PROGRAM MAIN
VAR
	power1:MC_Power;
	axis1: AXIS_REF;
	power1_do: BOOL;
	jog1:MC_Jog;
	jog_for: BOOL;
	jog_back: BOOL;
	
	//增加代码，与原版本程序做区分
	a:INT;
	b:INT;
	c:INT;
	d:INT;
	add1: FB_ADD;
END_VAR

power1(
	Axis:= axis1, 
	Enable:= power1_do, 
	Enable_Positive:= TRUE, 
	Enable_Negative:= TRUE, 
	Override:= , 
	BufferMode:= , 
	Options:= , 
	Status=> , 
	Busy=> , 
	Active=> , 
	Error=> , 
	ErrorID=> );
jog1(
	Axis:= axis1, 
	JogForward:= jog_for, 
	JogBackwards:= jog_back, 
	Mode:= , 
	Position:= , 
	Velocity:= , 
	Acceleration:= , 
	Deceleration:= , 
	Jerk:= , 
	Done=> , 
	Busy=> , 
	Active=> , 
	CommandAborted=> , 
	Error=> , 
	ErrorID=> );
	add1(in1:= a, in2:= b, in3:= c, out=>d );

END_PROGRAM

(* stored: Version 1.1.0.1, ProductVersion 3.1.4024.12
   POU MAIN: Id {8c4829e7-7c54-48b1-99ba-7f14b3668b23}, SpecialFunc None *)
